{attribute addProperty BoxType "EP2809-0042-0018"}
{attribute addProperty Id "DO_X01AT %Q*ARRAY[0..1] OF DO_X_7F374EB0429496728842949672950DO_X02AT %Q*ARRAY[0..1] OF DO_X_7F374EB0429496728842949672950DO_X03AT %Q*ARRAY[0..1] OF DO_X_7F374EB0429496728842949672950DO_X04AT %Q*ARRAY[0..1] OF DO_X_7F374EB0429496728842949672950DO_X05AT %Q*ARRAY[0..1] OF DO_X_7F374EB0429496728842949672950DO_X06AT %Q*ARRAY[0..1] OF DO_X_7F374EB0429496728842949672950DO_X07AT %Q*ARRAY[0..1] OF DO_X_7F374EB0429496728842949672950DO_X08AT %Q*ARRAY[0..1] OF DO_X_7F374EB0429496728842949672950WcStateAT %I*WcState_64F6A8C6810InfoDataAT %I*InfoData_192954DE1620"}
{attribute addProperty CRC "845911702"}
{attribute addProperty SizeInBites "4294967256"}
{attribute addProperty SizeInBytes "34359738363"}
TYPE EP2809_F05176C6 :
STRUCT
	{attribute addProperty Name "DO_X01"}
	DO_X01 : ARRAY[0..1] OF DO_X_7F374EB0;
	{attribute addProperty Name "DO_X02"}
	DO_X02 : ARRAY[0..1] OF DO_X_7F374EB0;
	{attribute addProperty Name "DO_X03"}
	DO_X03 : ARRAY[0..1] OF DO_X_7F374EB0;
	{attribute addProperty Name "DO_X04"}
	DO_X04 : ARRAY[0..1] OF DO_X_7F374EB0;
	{attribute addProperty Name "DO_X05"}
	DO_X05 : ARRAY[0..1] OF DO_X_7F374EB0;
	{attribute addProperty Name "DO_X06"}
	DO_X06 : ARRAY[0..1] OF DO_X_7F374EB0;
	{attribute addProperty Name "DO_X07"}
	DO_X07 : ARRAY[0..1] OF DO_X_7F374EB0;
	{attribute addProperty Name "DO_X08"}
	DO_X08 : ARRAY[0..1] OF DO_X_7F374EB0;
	{attribute addProperty Name "WcState"}
	WcState : WcState_64F6A8C6;
	{attribute addProperty Name "InfoData"}
	InfoData : InfoData_192954DE;
END_STRUCT
END_TYPE

(* stored: Version 1.2.0.0, ProductVersion 3.1.4024.9
   DUT EP2809_F05176C6: Id {d604a23a-08ae-4407-ab6c-5adcc37301ce} *)
